{attribute 'GeneratedUsingTerminal: EK1100-0000-0018'}
{attribute addProperty BoxType "EK1100-0000-0018"}
{attribute addProperty Id "Beckhoff_ELM3xxx_0030EK1122Beckhoff_ELM3xxx_0030EK1122_95B170302A_0001_ELM3002_0030_0017ELM3002_3D4ED79F42A_0002_ELM3002_0030_0018ELM3002_3D4ED79F42A_0003_ELM3004_0030_0018ELM3004_177D76D464A_0004_ELM3004_0030_0019ELM3004_177D76D464A_0005_ELM3502_0030_0019ELM3502_3D4ED79F42A_0006_ELM3504_0030_0019ELM3504_177D76D464"}
{attribute addProperty CRC "1322383127"}
{attribute addProperty Size "320"}
TYPE Beckhoff_ELM3xxx_0030_4ED1F717 EXTENDS EK1100_1FC0878B :
STRUCT
	{attribute addProperty Name "Beckhoff_ELM3xxx_0030EK1122"}
	{attribute addProperty PreviousPort "Beckhoff ELM3xxx-0030 : B"}
	Beckhoff_ELM3xxx_0030EK1122 : Beckhoff_ELM3xxx_0030EK1122_95B17030;
	{attribute addProperty Name "A_0001_ELM3002_0030_0017"}
	{attribute addProperty PreviousPort "Beckhoff ELM3xxx-0030EK1122 : C"}
	A_0001_ELM3002_0030_0017 : ELM3002_3D4ED79F;
	{attribute addProperty Name "A_0002_ELM3002_0030_0018"}
	{attribute addProperty PreviousPort "A_0001(ELM3002-0030-0017) : B"}
	A_0002_ELM3002_0030_0018 : ELM3002_3D4ED79F;
	{attribute addProperty Name "A_0003_ELM3004_0030_0018"}
	{attribute addProperty PreviousPort "A_0002(ELM3002-0030-0018) : B"}
	A_0003_ELM3004_0030_0018 : ELM3004_177D76D4;
	{attribute addProperty Name "A_0004_ELM3004_0030_0019"}
	{attribute addProperty PreviousPort "A_0003(ELM3004-0030-0018) : B"}
	A_0004_ELM3004_0030_0019 : ELM3004_177D76D4;
	{attribute addProperty Name "A_0005_ELM3502_0030_0019"}
	{attribute addProperty PreviousPort "A_0004(ELM3004-0030-0019) : B"}
	A_0005_ELM3502_0030_0019 : ELM3502_3D4ED79F;
	{attribute addProperty Name "A_0006_ELM3504_0030_0019"}
	{attribute addProperty PreviousPort "A_0005(ELM3502-0030-0019) : B"}
	A_0006_ELM3504_0030_0019 : ELM3504_177D76D4;
END_STRUCT
END_TYPE

(* stored: Version 1.2.0.0, ProductVersion 3.1.4024.9
   DUT Beckhoff_ELM3xxx_0030_4ED1F717: Id {0e59744e-4536-45e3-beb2-2cbc7c959d0c} *)
